(* CoDeSys 2.3.9.50 project: 4E.pr6 *)
(* Libraries: STANDARD.LB6 5.6.98 12:03:02 *)

(* POU MAIN, LD *)
PROGRAM MAIN
VAR
	CookieCounter AT %IX0.1: BOOL;
	C1: CTU;
	A AT %IX0.7: BOOL;
	OvenOn AT %QX0.0: BOOL;
	ClosetoOven AT %QX0.1: BOOL;
	removeCookies AT %IX0.2: BOOL;
	Indicator AT %QX0.3: BOOL;
END_VAR
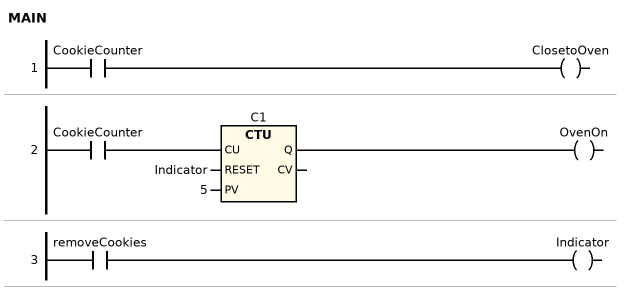
_LD_ (* Ladder Diagram *)
NETWORK 1
	[CookieCounter] --- (ClosetoOven)
NETWORK 2
	[CookieCounter] - C1:CTU(CU: *, RESET: Indicator, PV: 5) --- (OvenOn)
NETWORK 3
	[removeCookies] --- (Indicator)
_END_LD_
(* the same logic as Structured Text *)
(* Network 1 *)
ClosetoOven := CookieCounter;
(* Network 2 *)
C1(CU := CookieCounter, RESET := Indicator, PV := 5);
OvenOn := C1.Q;
(* Network 3 *)
Indicator := removeCookies;
END_PROGRAM
